TYPE ST_EbaraPTM EXTENDS ST_PTM :
STRUCT
(* Extension of the PTM archetype for Ebara turbo controllers 
Applicable to: 
ETC series
*)
//Controls
q_xStart   : BOOL; //Momentary start switch
q_xStop    : BOOL; //Momentary stop switch
q_xReset   : BOOL; //Momentary reset switch - resets protection functions
q_xProtection : BOOL; //NC. If opened, pump will decelerate/not start

i_xSpeedSetSW    : BOOL; //Request to set speed
q_xSpeedSetDO    : BOOL; //Momentary switch to program commanded speed
q_iSpeedSet   : DINT; //Requested speed (min. 100 RPM)

i_xOverride   : BOOL; //Override mode - ignores interlocks

//Readbacks - also has Accel/At speed/Decel/Fault/Cur Speed (min 100RPM)
i_xRotate : BOOL; //If open, pump is rotating
i_xDecel  : BOOL; //If closed, brake engaged (pump decelerating)
i_iRawSpeed	:	INT; //Raw pump speed from analog input

END_STRUCT
END_TYPE

(* stored: Version 1.1.0.1, ProductVersion 3.1.4018.5
   DUT ST_EbaraPTM: Id {00dd7679-7d3a-464d-8613-c714e423a1cf} *)
